FUNCTION_BLOCK VCylinder_HMI (* Service Interface Function Block Type *)
  (* Standard: 61499-2 *)
  (* Version 0.0, 9/14/2008, Horst Mayer, nxtControl GmbH, template *)
  PACKAGE Main;
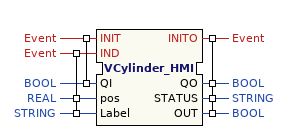
  EVENT_INPUT
    INIT WITH QI;
    IND WITH pos, Label;
  END_EVENT
  EVENT_OUTPUT
    INITO WITH QO, STATUS, OUT;
  END_EVENT
  VAR_INPUT
    QI : BOOL;
    pos : REAL;
    Label : STRING;
  END_VAR
  VAR_OUTPUT
    QO : BOOL; (* Event Output Qualifier *)
    STATUS : STRING; (* Service Status *)
    OUT : BOOL;
  END_VAR
END_FUNCTION_BLOCK
